/// This struct contains variables that
/// * are read from outside (e.g. HMI) to retrieve information about the unit's current state and (temporary) parameters (= `publish`) 
/// * are written from outside (e.g. HMI) to control the unit via ADS (= `subscribe`) 
TYPE HandlingCom :
STRUCT
  Publish : HandlingComPublish;
  Subscribe : HandlingComSubscribe;
END_STRUCT
END_TYPE

(* stored: Version 1.1.0.1
   DUT HandlingCom: Id {b5c6123a-8906-4352-aa22-fa09e637940b} *)
